// TwinCAT 3 PLC project PLC1
// ProgramVersion: 3.1.4023.0
// libraries:
//   Tc2_EtherCAT, * (Beckhoff Automation GmbH)
//   Tc2_MC2, * (Beckhoff Automation GmbH)
//   Tc2_MC2_Drive, * (Beckhoff Automation GmbH)
//   Tc2_Standard, * (Beckhoff Automation GmbH)
//   Tc2_System, * (Beckhoff Automation GmbH)
//   Tc2_Utilities, * (Beckhoff Automation GmbH)
//   Tc3_Module, * (Beckhoff Automation GmbH)
// project tree:
//   / PlcTask.TcTTO
//   POUs/ AxisBase.TcPOU, IO.TcPOU, MAIN.TcPOU, Recorder.TcPOU
// real-time tasks:
//   TASK PlcTask: cycle T#1ms, priority 20, ADS port 350
// motion (NC):
//   TASK NC-Task 1 SAF: cycle T#500us, priority 4, ADS port 501
//   TASK NC-Task 1 SVB: cycle T#1ms, priority 8, ADS port 511
//   AXIS motor_x1 (id 20)
//     OtherSettings: AllowMotionCmdToSlave=true, DataPersistence=true
//     encoder EncType=1
//     drive DrvType=5
//       Analog: TorqueSetpointScale=10, ScaleFactorActTorque=0.1
//       TimeComp: TaskDelayCycles=1
//     controller CtrType=1
//       CtrPara: PriorControlFactor=1
//         Observer: BandWidth=20
//   AXIS motor_x0 (id 1)
//     OtherSettings: AllowMotionCmdToSlave=true, DataPersistence=true
//     encoder EncType=1
//     drive DrvType=5
//       Analog: TorqueSetpointScale=10, ScaleFactorActTorque=0.1
//       TimeComp: TaskDelayCycles=1
//     controller CtrType=1
//       CtrPara: PriorControlFactor=1
//         Observer: BandWidth=20
//   AXIS motor_y0 (id 2)
//     OtherSettings: AllowMotionCmdToSlave=true, DataPersistence=true
//     encoder EncType=1
//     drive DrvType=5
//       Analog: TorqueSetpointScale=10, ScaleFactorActTorque=0.1
//       TimeComp: TaskDelayCycles=1
//     controller CtrType=1
//       CtrPara: PriorControlFactor=1
//         Observer: BandWidth=20
//   AXIS motor_y1 (id 3)
//     OtherSettings: AllowMotionCmdToSlave=true, DataPersistence=true
//     encoder EncType=1
//     drive DrvType=5
//       Analog: TorqueSetpointScale=10, ScaleFactorActTorque=0.1
//       TimeComp: TaskDelayCycles=1
//     controller CtrType=1
//       CtrPara: PriorControlFactor=1
//         Observer: BandWidth=20
//   AXIS motor_z1 (id 21)
//     OtherSettings: AllowMotionCmdToSlave=true, DataPersistence=true
//     encoder EncType=1
//     drive DrvType=5
//       Analog: TorqueSetpointScale=10, ScaleFactorActTorque=0.1
//       TimeComp: TaskDelayCycles=1
//     controller CtrType=1
//       CtrPara: PriorControlFactor=1
//         Observer: BandWidth=20
//   AXIS motor_z0 (id 4)
//     OtherSettings: AllowMotionCmdToSlave=true, DataPersistence=true
//     encoder EncType=1
//     drive DrvType=5
//       Analog: TorqueSetpointScale=10, ScaleFactorActTorque=0.1
//       TimeComp: TaskDelayCycles=1
//     controller CtrType=1
//       CtrPara: PriorControlFactor=1
//         Observer: BandWidth=20
//   AXIS motor_a0 (id 5)
//     OtherSettings: AllowMotionCmdToSlave=true, DataPersistence=true
//     encoder EncType=1
//     drive DrvType=5
//       Analog: TorqueSetpointScale=10, ScaleFactorActTorque=0.1
//       TimeComp: TaskDelayCycles=1
//     controller CtrType=1
//       CtrPara: PriorControlFactor=1
//         Observer: BandWidth=20
//   AXIS motor_b0 (id 6)
//     OtherSettings: AllowMotionCmdToSlave=true, DataPersistence=true
//     encoder EncType=1
//     drive DrvType=5
//       Analog: TorqueSetpointScale=10, ScaleFactorActTorque=0.1
//       TimeComp: TaskDelayCycles=1
//     controller CtrType=1
//       CtrPara: PriorControlFactor=1
//         Observer: BandWidth=20
//   AXIS motor_c0 (id 7)
//     OtherSettings: AllowMotionCmdToSlave=true, DataPersistence=true
//     encoder EncType=1
//     drive DrvType=5
//       Analog: TorqueSetpointScale=10, ScaleFactorActTorque=0.1
//       TimeComp: TaskDelayCycles=1
//     controller CtrType=1
//       CtrPara: PriorControlFactor=1
//         Observer: BandWidth=20
//   AXIS motor_d0 (id 8)
//     OtherSettings: AllowMotionCmdToSlave=true, DataPersistence=true
//     encoder EncType=1
//     drive DrvType=5
//       Analog: TorqueSetpointScale=10, ScaleFactorActTorque=0.1
//       TimeComp: TaskDelayCycles=1
//     controller CtrType=1
//       CtrPara: PriorControlFactor=1
//         Observer: BandWidth=20
//   AXIS motor_e0 (id 9)
//     OtherSettings: AllowMotionCmdToSlave=true, DataPersistence=true
//     encoder EncType=1
//     drive DrvType=5
//       Analog: TorqueSetpointScale=10, ScaleFactorActTorque=0.1
//       TimeComp: TaskDelayCycles=1
//     controller CtrType=1
//       CtrPara: PriorControlFactor=1
//         Observer: BandWidth=20
//   AXIS motor_x_master (id 10)
//     OtherSettings: AllowMotionCmdToSlave=true
//     encoder EncType=1
//     drive DrvType=5
//       Analog: TorqueSetpointScale=10, ScaleFactorActTorque=0.1
//       TimeComp: TaskDelayCycles=1
//     controller CtrType=1
//       CtrPara: PriorControlFactor=1
//         Observer: BandWidth=20
//   AXIS motor_y_master (id 11)
//     OtherSettings: AllowMotionCmdToSlave=true
//     encoder EncType=1
//     drive DrvType=5
//       Analog: TorqueSetpointScale=10, ScaleFactorActTorque=0.1
//       TimeComp: TaskDelayCycles=1
//     controller CtrType=1
//       CtrPara: PriorControlFactor=1
//         Observer: BandWidth=20
//   AXIS motor_z_master (id 12)
//     OtherSettings: AllowMotionCmdToSlave=true
//     encoder EncType=1
//     drive DrvType=5
//       Analog: TorqueSetpointScale=10, ScaleFactorActTorque=0.1
//       TimeComp: TaskDelayCycles=1
//     controller CtrType=1
//       CtrPara: PriorControlFactor=1
//         Observer: BandWidth=20
//   AXIS motor_a_master (id 13)
//     OtherSettings: AllowMotionCmdToSlave=true
//     encoder EncType=1
//     drive DrvType=5
//       Analog: TorqueSetpointScale=10, ScaleFactorActTorque=0.1
//       TimeComp: TaskDelayCycles=1
//     controller CtrType=1
//       CtrPara: PriorControlFactor=1
//         Observer: BandWidth=20
//   AXIS motor_b_master (id 14)
//     OtherSettings: AllowMotionCmdToSlave=true
//     encoder EncType=1
//     drive DrvType=5
//       Analog: TorqueSetpointScale=10, ScaleFactorActTorque=0.1
//       TimeComp: TaskDelayCycles=1
//     controller CtrType=1
//       CtrPara: PriorControlFactor=1
//         Observer: BandWidth=20
//   AXIS motor_c_master (id 15)
//     OtherSettings: AllowMotionCmdToSlave=true
//     encoder EncType=1
//     drive DrvType=5
//       Analog: TorqueSetpointScale=10, ScaleFactorActTorque=0.1
//       TimeComp: TaskDelayCycles=1
//     controller CtrType=1
//       CtrPara: PriorControlFactor=1
//         Observer: BandWidth=20
//   AXIS motor_d_master (id 16)
//     OtherSettings: AllowMotionCmdToSlave=true
//     encoder EncType=1
//     drive DrvType=5
//       Analog: TorqueSetpointScale=10, ScaleFactorActTorque=0.1
//       TimeComp: TaskDelayCycles=1
//     controller CtrType=1
//       CtrPara: PriorControlFactor=1
//         Observer: BandWidth=20
//   AXIS motor_e_master (id 17)
//     OtherSettings: AllowMotionCmdToSlave=true
//     encoder EncType=1
//     drive DrvType=5
//       Analog: TorqueSetpointScale=10, ScaleFactorActTorque=0.1
//       TimeComp: TaskDelayCycles=1
//     controller CtrType=1
//       CtrPara: PriorControlFactor=1
//         Observer: BandWidth=20
//   AXIS motor_z1_multimaster (id 22)
//     OtherSettings: AllowMotionCmdToSlave=true
//     encoder EncType=1
//     drive DrvType=5
//       Analog: TorqueSetpointScale=10, ScaleFactorActTorque=0.1
//       TimeComp: TaskDelayCycles=1
//     controller CtrType=1
//       CtrPara: PriorControlFactor=1
//         Observer: BandWidth=20
//   AXIS motor_z0_multimaster (id 18)
//     OtherSettings: AllowMotionCmdToSlave=true
//     encoder EncType=1
//     drive DrvType=5
//       Analog: TorqueSetpointScale=10, ScaleFactorActTorque=0.1
//       TimeComp: TaskDelayCycles=1
//     controller CtrType=1
//       CtrPara: PriorControlFactor=1
//         Observer: BandWidth=20
//   AXIS motor_z1_masterOffset (id 23)
//     OtherSettings: AllowMotionCmdToSlave=true
//     encoder EncType=1
//     drive DrvType=5
//       Analog: TorqueSetpointScale=10, ScaleFactorActTorque=0.1
//       TimeComp: TaskDelayCycles=1
//     controller CtrType=1
//       CtrPara: PriorControlFactor=1
//         Observer: BandWidth=20
//   AXIS motor_z0_masterOffset (id 19)
//     OtherSettings: AllowMotionCmdToSlave=true
//     encoder EncType=1
//     drive DrvType=5
//       Analog: TorqueSetpointScale=10, ScaleFactorActTorque=0.1
//       TimeComp: TaskDelayCycles=1
//     controller CtrType=1
//       CtrPara: PriorControlFactor=1
//         Observer: BandWidth=20
// variable links:
//   PLC1/PLC1 Instance <-> NC-Task 1 SAF/Axes/motor_a0
//     PlcTask Inputs/MAIN.motor_a0.axis.NcToPlc <-> Outputs/ToPlc
//     PlcTask Outputs/MAIN.motor_a0.axis.PlcToNc <-> Inputs/FromPlc
//   PLC1/PLC1 Instance <-> NC-Task 1 SAF/Axes/motor_a_master
//     PlcTask Inputs/MAIN.motor_a_master.axis.NcToPlc <-> Outputs/ToPlc
//     PlcTask Outputs/MAIN.motor_a_master.axis.PlcToNc <-> Inputs/FromPlc
//   PLC1/PLC1 Instance <-> NC-Task 1 SAF/Axes/motor_b0
//     PlcTask Inputs/MAIN.motor_b0.axis.NcToPlc <-> Outputs/ToPlc
//     PlcTask Outputs/MAIN.motor_b0.axis.PlcToNc <-> Inputs/FromPlc
//   PLC1/PLC1 Instance <-> NC-Task 1 SAF/Axes/motor_b_master
//     PlcTask Inputs/MAIN.motor_b_master.axis.NcToPlc <-> Outputs/ToPlc
//     PlcTask Outputs/MAIN.motor_b_master.axis.PlcToNc <-> Inputs/FromPlc
//   PLC1/PLC1 Instance <-> NC-Task 1 SAF/Axes/motor_c0
//     PlcTask Inputs/MAIN.motor_c0.axis.NcToPlc <-> Outputs/ToPlc
//     PlcTask Outputs/MAIN.motor_c0.axis.PlcToNc <-> Inputs/FromPlc
//   PLC1/PLC1 Instance <-> NC-Task 1 SAF/Axes/motor_c_master
//     PlcTask Inputs/MAIN.motor_c_master.axis.NcToPlc <-> Outputs/ToPlc
//     PlcTask Outputs/MAIN.motor_c_master.axis.PlcToNc <-> Inputs/FromPlc
//   PLC1/PLC1 Instance <-> NC-Task 1 SAF/Axes/motor_d0
//     PlcTask Inputs/MAIN.motor_d0.axis.NcToPlc <-> Outputs/ToPlc
//     PlcTask Outputs/MAIN.motor_d0.axis.PlcToNc <-> Inputs/FromPlc
//   PLC1/PLC1 Instance <-> NC-Task 1 SAF/Axes/motor_d_master
//     PlcTask Inputs/MAIN.motor_d_master.axis.NcToPlc <-> Outputs/ToPlc
//     PlcTask Outputs/MAIN.motor_d_master.axis.PlcToNc <-> Inputs/FromPlc
//   PLC1/PLC1 Instance <-> NC-Task 1 SAF/Axes/motor_e0
//     PlcTask Inputs/MAIN.motor_e0.axis.NcToPlc <-> Outputs/ToPlc
//     PlcTask Outputs/MAIN.motor_e0.axis.PlcToNc <-> Inputs/FromPlc
//   PLC1/PLC1 Instance <-> NC-Task 1 SAF/Axes/motor_e_master
//     PlcTask Inputs/MAIN.motor_e_master.axis.NcToPlc <-> Outputs/ToPlc
//     PlcTask Outputs/MAIN.motor_e_master.axis.PlcToNc <-> Inputs/FromPlc
//   PLC1/PLC1 Instance <-> NC-Task 1 SAF/Axes/motor_x0
//     PlcTask Inputs/MAIN.motor_x0.axis.NcToPlc <-> Outputs/ToPlc
//     PlcTask Outputs/MAIN.motor_x0.axis.PlcToNc <-> Inputs/FromPlc
//   PLC1/PLC1 Instance <-> NC-Task 1 SAF/Axes/motor_x1
//     PlcTask Inputs/MAIN.motor_x1.axis.NcToPlc <-> Outputs/ToPlc
//     PlcTask Outputs/MAIN.motor_x1.axis.PlcToNc <-> Inputs/FromPlc
//   PLC1/PLC1 Instance <-> NC-Task 1 SAF/Axes/motor_x_master
//     PlcTask Inputs/MAIN.motor_x_master.axis.NcToPlc <-> Outputs/ToPlc
//     PlcTask Outputs/MAIN.motor_x_master.axis.PlcToNc <-> Inputs/FromPlc
//   PLC1/PLC1 Instance <-> NC-Task 1 SAF/Axes/motor_y0
//     PlcTask Inputs/MAIN.motor_y0.axis.NcToPlc <-> Outputs/ToPlc
//     PlcTask Outputs/MAIN.motor_y0.axis.PlcToNc <-> Inputs/FromPlc
//   PLC1/PLC1 Instance <-> NC-Task 1 SAF/Axes/motor_y1
//     PlcTask Inputs/MAIN.motor_y1.axis.NcToPlc <-> Outputs/ToPlc
//     PlcTask Outputs/MAIN.motor_y1.axis.PlcToNc <-> Inputs/FromPlc
//   PLC1/PLC1 Instance <-> NC-Task 1 SAF/Axes/motor_y_master
//     PlcTask Inputs/MAIN.motor_y_master.axis.NcToPlc <-> Outputs/ToPlc
//     PlcTask Outputs/MAIN.motor_y_master.axis.PlcToNc <-> Inputs/FromPlc
//   PLC1/PLC1 Instance <-> NC-Task 1 SAF/Axes/motor_z0
//     PlcTask Inputs/MAIN.motor_z0.axis.NcToPlc <-> Outputs/ToPlc
//     PlcTask Outputs/MAIN.motor_z0.axis.PlcToNc <-> Inputs/FromPlc
//   PLC1/PLC1 Instance <-> NC-Task 1 SAF/Axes/motor_z0_masterOffset
//     PlcTask Inputs/MAIN.motor_z0_master_offset.axis.NcToPlc <-> Outputs/ToPlc
//     PlcTask Outputs/MAIN.motor_z0_master_offset.axis.PlcToNc <-> Inputs/FromPlc
//   PLC1/PLC1 Instance <-> NC-Task 1 SAF/Axes/motor_z0_multimaster
//     PlcTask Inputs/MAIN.motor_z0_multimaster.axis.NcToPlc <-> Outputs/ToPlc
//     PlcTask Outputs/MAIN.motor_z0_multimaster.axis.PlcToNc <-> Inputs/FromPlc
//   PLC1/PLC1 Instance <-> NC-Task 1 SAF/Axes/motor_z1
//     PlcTask Inputs/MAIN.motor_z1.axis.NcToPlc <-> Outputs/ToPlc
//     PlcTask Outputs/MAIN.motor_z1.axis.PlcToNc <-> Inputs/FromPlc
//   PLC1/PLC1 Instance <-> NC-Task 1 SAF/Axes/motor_z1_masterOffset
//     PlcTask Inputs/MAIN.motor_z1_master_offset.axis.NcToPlc <-> Outputs/ToPlc
//     PlcTask Outputs/MAIN.motor_z1_master_offset.axis.PlcToNc <-> Inputs/FromPlc
//   PLC1/PLC1 Instance <-> NC-Task 1 SAF/Axes/motor_z1_multimaster
//     PlcTask Inputs/MAIN.motor_z1_multimaster.axis.NcToPlc <-> Outputs/ToPlc
//     PlcTask Outputs/MAIN.motor_z1_multimaster.axis.PlcToNc <-> Inputs/FromPlc
//   PLC1/PLC1 Instance <-> NC-Task 1 SAF/Axes/motor_z_master
//     PlcTask Inputs/MAIN.motor_z_master.axis.NcToPlc <-> Outputs/ToPlc
//     PlcTask Outputs/MAIN.motor_z_master.axis.PlcToNc <-> Inputs/FromPlc

CONFIGURATION PLC1
    RESOURCE PLC ON TwinCAT3
        TASK PlcTask(INTERVAL := T#1ms, PRIORITY := 20);
        PROGRAM MAIN WITH PlcTask : MAIN;
    END_RESOURCE
END_CONFIGURATION

// ---- POUs/MAIN.TcPOU
PROGRAM MAIN
VAR
	//Variables of type AXIS_REF to your motors.
	//Add more motors if you need to.
	
	motor_x0 : AxisBase;
	motor_y0 : AxisBase;
	motor_z0 : AxisBase;
	motor_a0 : AxisBase;
	motor_b0 : AxisBase;
END_VAR

motor_x0();
motor_y0();
motor_z0();
motor_a0();
motor_b0();


IO();
Recorder();

END_PROGRAM

// ---- POUs/AxisBase.TcPOU
FUNCTION_BLOCK AxisBase
VAR_INPUT
END_VAR
VAR_OUTPUT

END_VAR
VAR
	axis : AXIS_REF;
	fbPower : MC_Power;
	bEnable : BOOL;
	bEnablePositiveMovement AT %I* : BOOL := TRUE; //Feed enable in positive direction.
	bEnableNegativeMovement AT %I* : BOOL := TRUE; //Feed enable in negative direction.
	
	fbHome : MC_Home;
	AxisHomed : BOOL;
	
	fbSoeReset: FB_SoEReset;

	pActPosAdress : POINTER TO LREAL := 0;
END_VAR


axis.ReadStatus();


	
fbPower(
	Axis:= axis, 
	Enable:= bEnable, //AND IO.EMCOK, 
	Enable_Positive:= bEnablePositiveMovement, 
	Enable_Negative:= bEnableNegativeMovement, 
	Override:= 100, 
	BufferMode:= ,
	Options:= , 
	Status=> , 
	Busy=> , 
	Active=> , 
	Error=> , 
	ErrorID=> );
	

fbHome(
	Axis:= axis, 
	Execute:= , 
	Position:= , 
	HomingMode:= MC_HomingMode.MC_Direct, 
	BufferMode:= , 
	Options:= , 
	bCalibrationCam:= , 
	Done=> , 
	Busy=> , 
	Active=> , 
	CommandAborted=> , 
	Error=> , 
	ErrorID=> );
	
	


IF fbSoeReset.Execute AND fbSoeReset.Busy THEN
	fbSoeReset.Execute := FALSE;
END_IF

fbSOEReset(
	Axis:= axis , 
	NetId:= , 
	Execute:= , 
	Timeout:= , 
	Busy=> , 
	Error=> , 
	AdsErrId=> , 
	SercosErrId=> );
	

IF(pActPosAdress = 0) THEN
	pActPosAdress := ADR(axis.NcToPlc.ActPos);
END_IF

END_FUNCTION_BLOCK

// ---- POUs/IO.TcPOU
PROGRAM IO
VAR
	//Link you hardware IO to these variables.
	//You can rename these variables as you like.
	DI1 AT %I* : BOOL;
	DI2 AT %I* : BOOL;	
	DI3 AT %I* : BOOL;
	DI4 AT %I* : BOOL;	
	DI5 AT %I* : BOOL;	
	DI6 AT %I* : BOOL;
	DI7 AT %I* : BOOL;	
	DI8 AT %I* : BOOL;	
	DI9 AT %I* : BOOL;
	DI10 AT %I* : BOOL;
	DI11 AT %I* : BOOL;
	DI12 AT %I* : BOOL;
	DI13 AT %I* : BOOL;
	DI14 AT %I* : BOOL;
	DI15 AT %I* : BOOL;
	DI16 AT %I* : BOOL;

	
	DO1 AT %Q* : BOOL;
	DO2 AT %Q* : BOOL;
	DO3 AT %Q* : BOOL;
	DO4 AT %Q* : BOOL;
	DO5 AT %Q* : BOOL;
	DO6 AT %Q* : BOOL;
	DO7 AT %Q* : BOOL;	
	
	AI1 AT %I* : INT;
	AI2 AT %I* : INT;
	AI3 AT %I* : INT;
	
	AO1 AT %Q* : INT;
	AO2 AT %Q* : INT;
	AO3 AT %Q* : INT;

	EMCOK  AT %I*:BOOL; //Emergency stop OK.
END_VAR

END_PROGRAM

// ---- POUs/Recorder.TcPOU
PROGRAM Recorder
VAR
	bRunning 	: BOOL;
	bGetValues 	: BOOL; //Signal from HMI that we want to read the saved values.
	//bRecord5axis : BOOL;
	
	

	nArrayIndex : INT;
	nEntryCount : INT; //How many entries exist for HMI to fetch.
	aPositions	: ARRAY[0..2048] OF LREAL;
	aCopy		: ARRAY[0..2048] OF LREAL; //HMI will fetch from aCopy and we can continue filling aPositions with new data.
	
	nIter		: INT;
	nIterMax 	: INT;
	
	//We don't know what motors the user will or will not have.
	//So IGEMS CNC sets these pointers to the adress of the motor position it wants to record.
	pAdresses : ARRAY[0..5] OF POINTER TO LREAL;
END_VAR

IF bGetValues	THEN //Signal that HMI is ready to copy values. Copy values to a second array that HMI can read from.
	nEntryCount := nArrayIndex;
	nArrayIndex := 0;
	
	MEMCPY(destAddr:= ADR(aCopy), srcAddr:= ADR(aPositions), n:= INT_TO_UDINT(8 * nEntryCount)); 
	bGetValues := FALSE;
END_IF


IF NOT bRunning THEN
	nArrayIndex := 0;
	RETURN;
END_IF



IF (nArrayIndex > 2048) THEN
	nArrayIndex := 0; //Wrapover if no one fetched the stored values.
END_IF



FOR nIter := 0 TO nIterMax DO
	//Get the act pos value.
	IF (pAdresses[nIter] <> 0) THEN 
		aPositions[nArrayIndex] := pAdresses[nIter]^; //Valid pointer has been set by over ADS, dereference it.
	ELSE 
		aPositions[nArrayIndex] := 0.0; //Not a valid pointer, just set the actual postion to 0.0
	END_IF
	
	nArrayIndex := nArrayIndex + 1;  
END_FOR;

END_PROGRAM
